// TIA Portal V19 export
TYPE "CoilHandling_Config"
   STRUCT
      SensorsDelayOn : Time := T#500ms;
      SensorsDelayOff : Time := T#500ms;
      CoilDiameterSetLoopSynchro : Real := 510.0;
      CoilDiameterRstLoopSynchro : Real := 600.0;
      MatCounter_Exist : Bool := TRUE;
   END_STRUCT;
END_TYPE
